FUNCTION_BLOCK ConfigurationManagerC
  (* Standard: 61499-2 *)
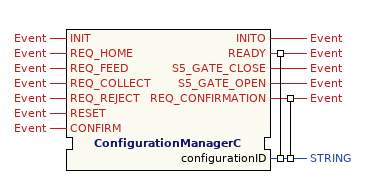
  EVENT_INPUT
    INIT;
    REQ_HOME;
    REQ_FEED;
    REQ_COLLECT;
    REQ_REJECT;
    RESET;
    CONFIRM;
  END_EVENT
  EVENT_OUTPUT
    INITO;
    READY WITH configurationID;
    S5_GATE_CLOSE;
    S5_GATE_OPEN;
    REQ_CONFIRMATION WITH configurationID;
  END_EVENT
  VAR_OUTPUT
    configurationID : STRING;
  END_VAR
  FBS
    FB1 : ConfigurationManager;
    FB2 : RobotinoViewUdp;
    FB3 : E_DELAY;
  END_FBS
  EVENT_CONNECTIONS
    INIT TO FB3.START;
    REQ_HOME TO FB1.REQ_HOME;
    REQ_FEED TO FB1.REQ_FEED;
    REQ_COLLECT TO FB1.REQ_COLLECT;
    REQ_REJECT TO FB1.REQ_REJECT;
    FB1.INITO TO INITO;
    FB1.READY TO READY;
    FB1.S5_GATE_CLOSE TO S5_GATE_CLOSE;
    FB1.S5_GATE_OPEN TO S5_GATE_OPEN;
    FB2.INITO TO FB1.INIT;
    FB1.CNF TO FB2.REQ;
    FB2.CNF TO FB1.REQ;
    FB3.EO TO FB2.INIT;
    INIT TO FB2.INIT;
    RESET TO FB1.RESET;
    FB1.REQ_CONFIRMATION TO REQ_CONFIRMATION;
    CONFIRM TO FB1.CONFIRM;
  END_CONNECTIONS
  DATA_CONNECTIONS
    FB2.dock_out TO FB1.robotinoPos;
    FB1.configurationID TO FB2.dock_in;
    FB1.configurationID TO configurationID;
  END_CONNECTIONS
END_FUNCTION_BLOCK
